{attribute 'qualified_only'}
{attribute 'strict'}
{attribute 'to_string'}
TYPE E_BaseEvents_Action :
(
	Start 		:= 0,
	Stop		:= 1,
	Confirm		:= 2
);
END_TYPE

(* stored: Version 1.1.0.1
   DUT E_BaseEvents_Action: Id {3afb22dd-47b4-4124-8e7b-ade6253ee77e} *)
